// TIA Portal project "Trạm 4" (V17)

(* hardware
DEVICE "S7-1200 station_1"  S7-1200 Station
   slot 0: "Rack_0"  S7-1200 Rack  Rack  V1.0
   slot 1: "PLC_1"  CPU 1214C DC/DC/DC  6ES7 214-1AG40-0XB0  V4.4
*)

// ===== PLC "PLC_1"  CPU 1214C DC/DC/DC =====

VAR_GLOBAL   // PLC tag table "Default tag table"
   "Cảm biến phôi" AT %I0.0 : Bool;
   "Cảm biến vị trí gắp vật" AT %I0.1 : Bool;
   "Cảm biến vị trí trạm sau" AT %I0.2 : Bool;
   "Cảm biến vị trí khay" AT %I0.3 : Bool;
   "Cảm biến tay gắp xuống" AT %I0.4 : Bool;
   "Cảm biến tay gắp lên" AT %I0.5 : Bool;
   "CB_Mau" AT %I0.6 : Bool;
   "CB_TramIn" AT %I0.7 : Bool;
   "Start" AT %I1.0 : Bool;
   "Stop" AT %I1.1 : Bool;
   "Auto" AT %I1.2 : Bool;
   "Reset" AT %I1.3 : Bool;
   "HTTRai" AT %Q0.0 : Bool;
   "HTPhai" AT %Q0.1 : Bool;
   "Xi lanh xuống" AT %Q0.2 : Bool;
   "Kẹp phôi" AT %Q0.3 : Bool;
   "Yêu cầu cấp phôi" AT %Q0.7 : Bool;
   "LedStart" AT %Q1.0 : Bool;
   "LedReset" AT %Q1.1 : Bool;
   "TG_Start" AT %M0.0 : Bool;
   "TG_HTVat" AT %M0.1 : Bool;
   "TG_HTVat2" AT %M0.2 : Bool;
   "TG_TayGapXuong" AT %M0.3 : Bool;
   "TG_DungNhaVat" AT %M1.0 : Bool;
   "TG_CoVat" AT %M1.1 : Bool;
   "TG_Khay3" AT %M0.6 : Bool;
   "TG_HTkhay2" AT %M9.0 : Bool;
   "TG_CBHTV" AT %M9.1 : Bool;
   "TGCBVat" AT %M10.0 : Bool;
   "TG_ChoKep" AT %M0.4 : Bool;
   "TG_XilanhLen" AT %M0.5 : Bool;
   "TG_TramTiep" AT %M0.7 : Bool;
   "TG_XuongGapVat" AT %M1.2 : Bool;
   "TG_KepVat" AT %M1.3 : Bool;
   "TG_HTPhai" AT %M1.4 : Bool;
   "TG_DungTraVat" AT %M1.5 : Bool;
   "TG_NhaVat" AT %M1.6 : Bool;
   "TG_NhaVat2" AT %M1.7 : Bool;
   "TG_GapLoi" AT %M2.0 : Bool;
   "TG_Button_Reset" AT %M3.0 : Bool;
   "Tag_1" AT %M3.1 : Bool;
   "Tag_2" AT %M3.2 : Bool;
   "Tag_3" AT %M3.3 : Bool;
   "Tag_4" AT %M3.4 : Bool;
   "Tag_5" AT %M5.0 : Bool;
   "Tag_6" AT %M5.1 : Bool;
   "TG_Start_Manual" AT %M2.1 : Bool;
   "TG_Start_Auto" AT %M2.2 : Bool;
   "TG_TruyenThong_Reset" AT %M2.3 : Bool;
   "Reset_Truyen" AT %M2.4 : Bool;
END_VAR

VAR_GLOBAL   // PLC tag table "Trung gian tin hieu truyen nhan"
   "TG_PhoiThap" AT %M4.0 : Bool;
   "TG_PhoiCao" AT %M4.1 : Bool;
END_VAR

DATA_BLOCK "Data_TruyenThong05"   // DB31
{ S7_Optimized_Access := 'FALSE' }
VERSION : 0.1
   VAR
      Nhan_1 : Bool;
      Nhan_2 : Bool;
      Nhan_3 : Bool;
      Nhan_4 : Bool;
      Nhan_5 : Bool;
      Nhan_6 : Bool;
      Nhan_7 : Bool;
      Nhan_8 : Bool;
      truyen_1 : Bool;
      truyen_2 : Bool;
      truyen_3 : Bool;
      truyen_4 : Bool;
      truyen_5 : Bool;
      truyen_6 : Bool;
      truyen_7 : Bool;
      truyen_8 : Bool;
      truyen_9 : Bool;
      truyen_10 : Bool;
      truyen_11 : Bool;
      truyen_12 : Bool;
      truyen_13 : Bool;
      truyen_14 : Bool;
      truyen_15 : Bool;
      truyen_16 : Bool;
   END_VAR
BEGIN
END_DATA_BLOCK

// folder: System blocks/Program resources

DATA_BLOCK "Cho_Kep"   // DB26
{ S7_Optimized_Access := 'TRUE' }
AUTHOR : Simatic
FAMILY : IEC
NAME : IEC_TMR
VERSION : 1.0
// stored: InstanceOfName IEC_TIMER
"IEC_TIMER"
BEGIN
END_DATA_BLOCK

DATA_BLOCK "DungTraVat"   // DB27
{ S7_Optimized_Access := 'TRUE' }
AUTHOR : Simatic
FAMILY : IEC
NAME : IEC_TMR
VERSION : 1.0
// stored: InstanceOfName IEC_TIMER
"IEC_TIMER"
BEGIN
END_DATA_BLOCK

DATA_BLOCK "IEC_Timer_0_DB"   // DB28
{ S7_Optimized_Access := 'TRUE' }
AUTHOR : Simatic
FAMILY : IEC
NAME : IEC_TMR
VERSION : 1.0
// stored: InstanceOfName IEC_TIMER
"IEC_TIMER"
BEGIN
END_DATA_BLOCK

DATA_BLOCK "NhaVat_1"   // DB29
{ S7_Optimized_Access := 'TRUE' }
AUTHOR : Simatic
FAMILY : IEC
NAME : IEC_TMR
VERSION : 1.0
// stored: InstanceOfName IEC_TIMER
"IEC_TIMER"
BEGIN
END_DATA_BLOCK

DATA_BLOCK "TIme_GapVat"   // DB30
{ S7_Optimized_Access := 'TRUE' }
AUTHOR : Simatic
FAMILY : IEC
NAME : IEC_TMR
VERSION : 1.0
// stored: InstanceOfName IEC_TIMER
"IEC_TIMER"
BEGIN
END_DATA_BLOCK

// folder: (top level)

FUNCTION "GapVat" : Void   // FC1, LAD
{ S7_Optimized_Access := 'TRUE' }
VERSION : 0.1
BEGIN

REGION Network 1: Xác định có phôi ( Done ) -> CB phát hiện phôi + tay gắp ở vị trí trên + tay kẹp chưa kẹp = TG có phôi.
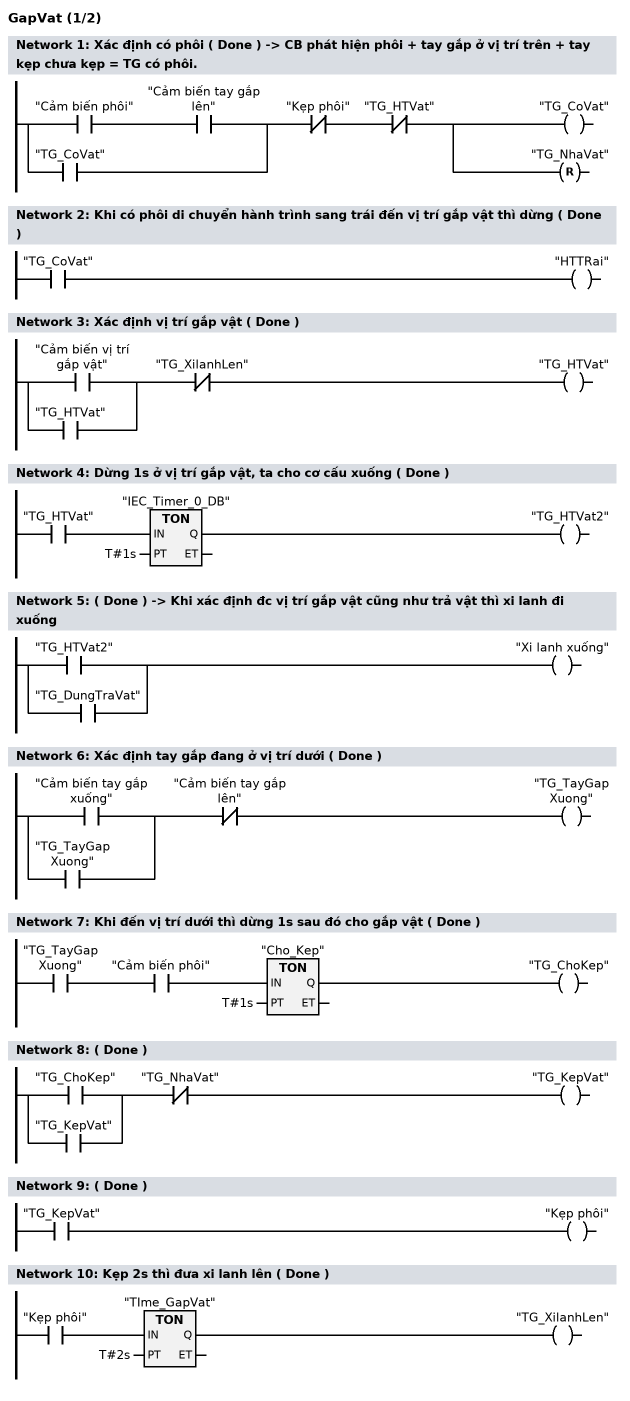
   RUNG wire#powerrail
      Contact( "Cảm biến phôi" )
      Contact( "Cảm biến tay gắp lên" )
      wire#w1
      I_Contact( "Kẹp phôi" )
      I_Contact( "TG_HTVat" )
      wire#w2
      Coil( "TG_CoVat" )
   END_RUNG
   RUNG wire#powerrail
      Contact( "TG_CoVat" )
   END_RUNG wire#w1
   RUNG wire#w2
      R_Coil( "TG_NhaVat" )
   END_RUNG
   // the same network as SCL:
   "TG_CoVat" := (("Cảm biến phôi" AND "Cảm biến tay gắp lên") OR "TG_CoVat") AND NOT "Kẹp phôi" AND NOT "TG_HTVat";
   IF "TG_CoVat" THEN "TG_NhaVat" := FALSE; END_IF;
END_REGION

REGION Network 2: Khi có phôi di chuyển hành trình sang trái đến vị trí gắp vật thì dừng ( Done )
   RUNG wire#powerrail
      Contact( "TG_CoVat" )
      Coil( "HTTRai" )
   END_RUNG
   // the same network as SCL:
   "HTTRai" := "TG_CoVat";
END_REGION

REGION Network 3: Xác định vị trí gắp vật ( Done )
   RUNG wire#powerrail
      Contact( "Cảm biến vị trí gắp vật" )
      wire#w1
      I_Contact( "TG_XilanhLen" )
      Coil( "TG_HTVat" )
   END_RUNG
   RUNG wire#powerrail
      Contact( "TG_HTVat" )
   END_RUNG wire#w1
   // the same network as SCL:
   "TG_HTVat" := ("Cảm biến vị trí gắp vật" OR "TG_HTVat") AND NOT "TG_XilanhLen";
END_REGION

REGION Network 4: Dừng 1s ở vị trí gắp vật, ta cho cơ cấu xuống ( Done )
   "IEC_Timer_0_DB".TON(IN := "TG_HTVat", PT := T#1s);
   "TG_HTVat2" := "IEC_Timer_0_DB".Q;
END_REGION

REGION Network 5: ( Done ) -> Khi xác định đc vị trí gắp vật cũng như trả vật thì xi lanh đi xuống
   RUNG wire#powerrail
      Contact( "TG_HTVat2" )
      wire#w1
      Coil( "Xi lanh xuống" )
   END_RUNG
   RUNG wire#powerrail
      Contact( "TG_DungTraVat" )
   END_RUNG wire#w1
   // the same network as SCL:
   "Xi lanh xuống" := "TG_HTVat2" OR "TG_DungTraVat";
END_REGION

REGION Network 6: Xác định tay gắp đang ở vị trí dưới ( Done )
   RUNG wire#powerrail
      Contact( "Cảm biến tay gắp xuống" )
      wire#w1
      I_Contact( "Cảm biến tay gắp lên" )
      Coil( "TG_TayGapXuong" )
   END_RUNG
   RUNG wire#powerrail
      Contact( "TG_TayGapXuong" )
   END_RUNG wire#w1
   // the same network as SCL:
   "TG_TayGapXuong" := ("Cảm biến tay gắp xuống" OR "TG_TayGapXuong") AND NOT "Cảm biến tay gắp lên";
END_REGION

REGION Network 7: Khi đến vị trí dưới thì dừng 1s sau đó cho gắp vật ( Done )
   "Cho_Kep".TON(IN := "TG_TayGapXuong" AND "Cảm biến phôi", PT := T#1s);
   "TG_ChoKep" := "Cho_Kep".Q;
END_REGION

REGION Network 8: ( Done )
   RUNG wire#powerrail
      Contact( "TG_ChoKep" )
      wire#w1
      I_Contact( "TG_NhaVat" )
      Coil( "TG_KepVat" )
   END_RUNG
   RUNG wire#powerrail
      Contact( "TG_KepVat" )
   END_RUNG wire#w1
   // the same network as SCL:
   "TG_KepVat" := ("TG_ChoKep" OR "TG_KepVat") AND NOT "TG_NhaVat";
END_REGION

REGION Network 9: ( Done )
   RUNG wire#powerrail
      Contact( "TG_KepVat" )
      Coil( "Kẹp phôi" )
   END_RUNG
   // the same network as SCL:
   "Kẹp phôi" := "TG_KepVat";
END_REGION

REGION Network 10: Kẹp 2s thì đưa xi lanh lên ( Done )
   "TIme_GapVat".TON(IN := "Kẹp phôi", PT := T#2s);
   "TG_XilanhLen" := "TIme_GapVat".Q;
END_REGION

REGION Network 11: Khi xi lanh ở vị tri trên và đang kẹp vật thì cho sang phải ( Done )
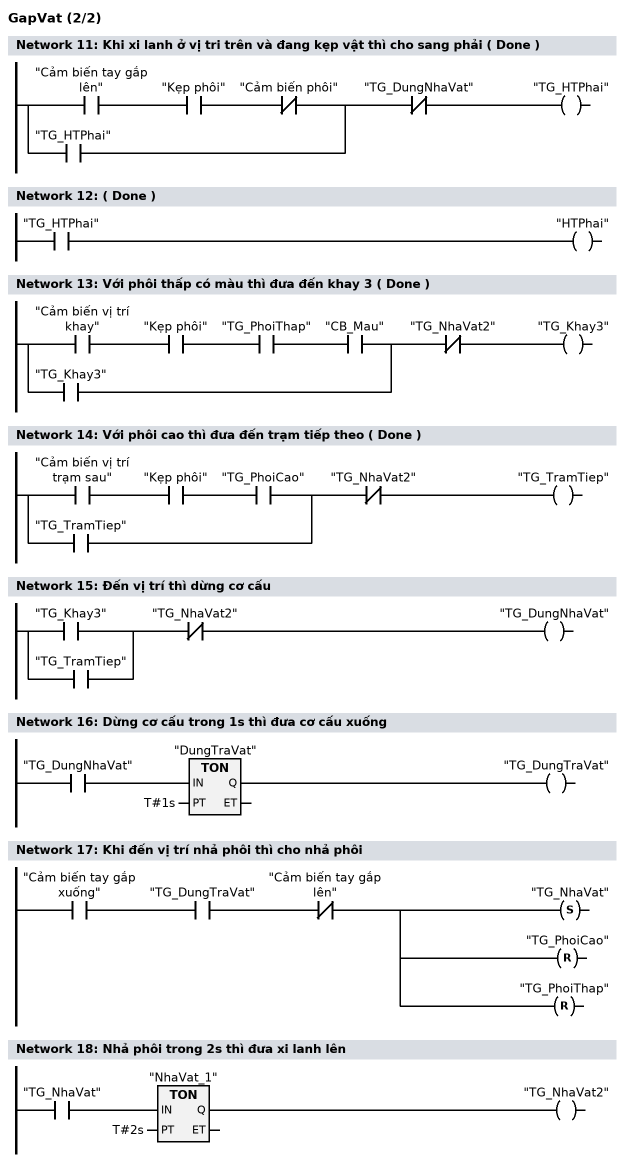
   RUNG wire#powerrail
      Contact( "Cảm biến tay gắp lên" )
      Contact( "Kẹp phôi" )
      I_Contact( "Cảm biến phôi" )
      wire#w1
      I_Contact( "TG_DungNhaVat" )
      Coil( "TG_HTPhai" )
   END_RUNG
   RUNG wire#powerrail
      Contact( "TG_HTPhai" )
   END_RUNG wire#w1
   // the same network as SCL:
   "TG_HTPhai" := (("Cảm biến tay gắp lên" AND "Kẹp phôi" AND NOT "Cảm biến phôi") OR "TG_HTPhai") AND NOT "TG_DungNhaVat";
END_REGION

REGION Network 12: ( Done )
   RUNG wire#powerrail
      Contact( "TG_HTPhai" )
      Coil( "HTPhai" )
   END_RUNG
   // the same network as SCL:
   "HTPhai" := "TG_HTPhai";
END_REGION

REGION Network 13: Với phôi thấp có màu thì đưa đến khay 3 ( Done )
   RUNG wire#powerrail
      Contact( "Cảm biến vị trí khay" )
      Contact( "Kẹp phôi" )
      Contact( "TG_PhoiThap" )
      Contact( "CB_Mau" )
      wire#w1
      I_Contact( "TG_NhaVat2" )
      Coil( "TG_Khay3" )
   END_RUNG
   RUNG wire#powerrail
      Contact( "TG_Khay3" )
   END_RUNG wire#w1
   // the same network as SCL:
   "TG_Khay3" := (("Cảm biến vị trí khay" AND "Kẹp phôi" AND "TG_PhoiThap" AND "CB_Mau") OR "TG_Khay3") AND NOT "TG_NhaVat2";
END_REGION

REGION Network 14: Với phôi cao thì đưa đến trạm tiếp theo ( Done )
   RUNG wire#powerrail
      Contact( "Cảm biến vị trí trạm sau" )
      Contact( "Kẹp phôi" )
      Contact( "TG_PhoiCao" )
      wire#w1
      I_Contact( "TG_NhaVat2" )
      Coil( "TG_TramTiep" )
   END_RUNG
   RUNG wire#powerrail
      Contact( "TG_TramTiep" )
   END_RUNG wire#w1
   // the same network as SCL:
   "TG_TramTiep" := (("Cảm biến vị trí trạm sau" AND "Kẹp phôi" AND "TG_PhoiCao") OR "TG_TramTiep") AND NOT "TG_NhaVat2";
END_REGION

REGION Network 15: Đến vị trí thì dừng cơ cấu
   RUNG wire#powerrail
      Contact( "TG_Khay3" )
      wire#w1
      I_Contact( "TG_NhaVat2" )
      Coil( "TG_DungNhaVat" )
   END_RUNG
   RUNG wire#powerrail
      Contact( "TG_TramTiep" )
   END_RUNG wire#w1
   // the same network as SCL:
   "TG_DungNhaVat" := ("TG_Khay3" OR "TG_TramTiep") AND NOT "TG_NhaVat2";
END_REGION

REGION Network 16: Dừng cơ cấu trong 1s thì đưa cơ cấu xuống
   "DungTraVat".TON(IN := "TG_DungNhaVat", PT := T#1s);
   "TG_DungTraVat" := "DungTraVat".Q;
END_REGION

REGION Network 17: Khi đến vị trí nhả phôi thì cho nhả phôi
   RUNG wire#powerrail
      Contact( "Cảm biến tay gắp xuống" )
      Contact( "TG_DungTraVat" )
      I_Contact( "Cảm biến tay gắp lên" )
      wire#w1
      S_Coil( "TG_NhaVat" )
   END_RUNG
   RUNG wire#w1
      R_Coil( "TG_PhoiCao" )
   END_RUNG
   RUNG wire#w1
      R_Coil( "TG_PhoiThap" )
   END_RUNG
   // the same network as SCL:
   IF "Cảm biến tay gắp xuống" AND "TG_DungTraVat" AND NOT "Cảm biến tay gắp lên" THEN
       "TG_NhaVat" := TRUE;
       "TG_PhoiCao" := FALSE;
       "TG_PhoiThap" := FALSE;
   END_IF;
END_REGION

REGION Network 18: Nhả phôi trong 2s thì đưa xi lanh lên
   "NhaVat_1".TON(IN := "TG_NhaVat", PT := T#2s);
   "TG_NhaVat2" := "NhaVat_1".Q;
END_REGION
END_FUNCTION

FUNCTION "OBReset" : Void   // FC2, LAD
{ S7_Optimized_Access := 'TRUE' }
VERSION : 0.1
   VAR_TEMP   // added for the SCL form of the ladder/FBD networks
      _w1 : Bool;
   END_VAR
BEGIN

REGION Network 1: Reset các trạng thái
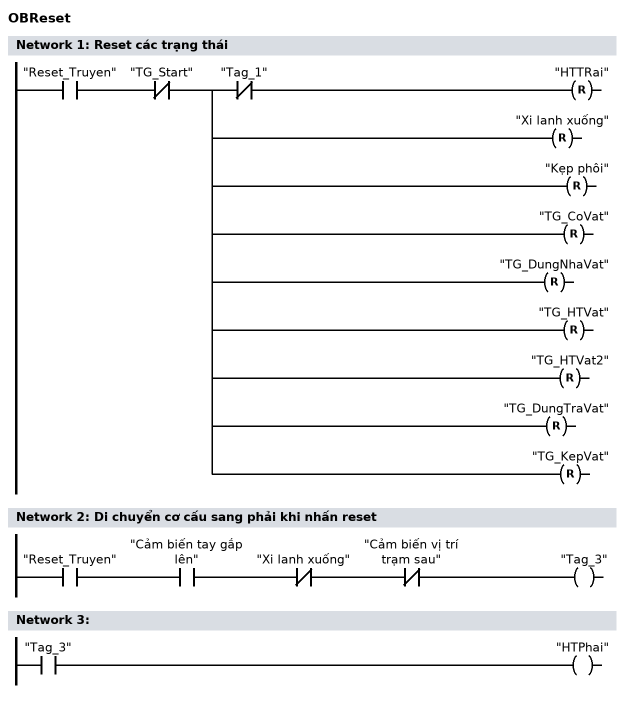
   RUNG wire#powerrail
      Contact( "Reset_Truyen" )
      I_Contact( "TG_Start" )
      wire#w1
      I_Contact( "Tag_1" )
      R_Coil( "HTTRai" )
   END_RUNG
   RUNG wire#w1
      R_Coil( "Xi lanh xuống" )
   END_RUNG
   RUNG wire#w1
      R_Coil( "Kẹp phôi" )
   END_RUNG
   RUNG wire#w1
      R_Coil( "TG_CoVat" )
   END_RUNG
   RUNG wire#w1
      R_Coil( "TG_DungNhaVat" )
   END_RUNG
   RUNG wire#w1
      R_Coil( "TG_HTVat" )
   END_RUNG
   RUNG wire#w1
      R_Coil( "TG_HTVat2" )
   END_RUNG
   RUNG wire#w1
      R_Coil( "TG_DungTraVat" )
   END_RUNG
   RUNG wire#w1
      R_Coil( "TG_KepVat" )
   END_RUNG
   // the same network as SCL:
   #_w1 := "Reset_Truyen" AND NOT "TG_Start";
   IF #_w1 AND NOT "Tag_1" THEN "HTTRai" := FALSE; END_IF;
   IF #_w1 THEN
       "Xi lanh xuống" := FALSE;
       "Kẹp phôi" := FALSE;
       "TG_CoVat" := FALSE;
       "TG_DungNhaVat" := FALSE;
       "TG_HTVat" := FALSE;
       "TG_HTVat2" := FALSE;
       "TG_DungTraVat" := FALSE;
       "TG_KepVat" := FALSE;
   END_IF;
END_REGION

REGION Network 2: Di chuyển cơ cấu sang phải khi nhấn reset
   RUNG wire#powerrail
      Contact( "Reset_Truyen" )
      Contact( "Cảm biến tay gắp lên" )
      I_Contact( "Xi lanh xuống" )
      I_Contact( "Cảm biến vị trí trạm sau" )
      Coil( "Tag_3" )
   END_RUNG
   // the same network as SCL:
   "Tag_3" := "Reset_Truyen" AND "Cảm biến tay gắp lên" AND NOT "Xi lanh xuống" AND NOT "Cảm biến vị trí trạm sau";
END_REGION

REGION Network 3
   RUNG wire#powerrail
      Contact( "Tag_3" )
      Coil( "HTPhai" )
   END_RUNG
   // the same network as SCL:
   "HTPhai" := "Tag_3";
END_REGION
END_FUNCTION

ORGANIZATION_BLOCK "Main"   // OB1, LAD, ProgramCycle
TITLE = "Main Program Sweep (Cycle)"
{ S7_Optimized_Access := 'TRUE' }
VERSION : 0.1
   VAR_INPUT
      Initial_Call : Bool;   // Initial call of this OB
      Remanence : Bool;   // =True, if remanent data are available
   END_VAR
BEGIN

REGION Network 1: Trạng thái Start ở chế độ Manual ( Done ) -> Vặn khóa + ấn Start và k có tín hiệu Auto từ HMI = Manual
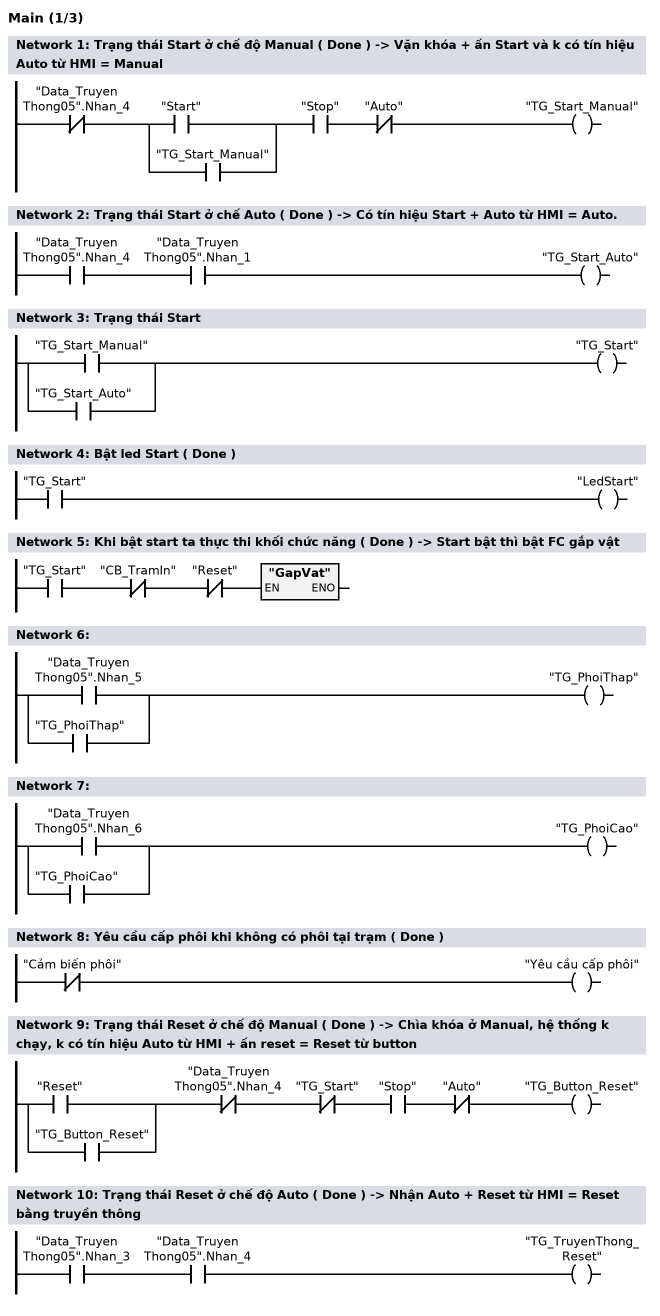
   RUNG wire#powerrail
      I_Contact( "Data_TruyenThong05".Nhan_4 )
      wire#w1
      Contact( "Start" )
      wire#w2
      Contact( "Stop" )
      I_Contact( "Auto" )
      Coil( "TG_Start_Manual" )
   END_RUNG
   RUNG wire#w1
      Contact( "TG_Start_Manual" )
   END_RUNG wire#w2
   // the same network as SCL:
   "TG_Start_Manual" := NOT "Data_TruyenThong05".Nhan_4 AND ("Start" OR "TG_Start_Manual") AND "Stop" AND NOT "Auto";
END_REGION

REGION Network 2: Trạng thái Start ở chế Auto ( Done ) -> Có tín hiệu Start + Auto từ HMI = Auto.
   RUNG wire#powerrail
      Contact( "Data_TruyenThong05".Nhan_4 )
      Contact( "Data_TruyenThong05".Nhan_1 )
      Coil( "TG_Start_Auto" )
   END_RUNG
   // the same network as SCL:
   "TG_Start_Auto" := "Data_TruyenThong05".Nhan_4 AND "Data_TruyenThong05".Nhan_1;
END_REGION

REGION Network 3: Trạng thái Start
   RUNG wire#powerrail
      Contact( "TG_Start_Manual" )
      wire#w1
      Coil( "TG_Start" )
   END_RUNG
   RUNG wire#powerrail
      Contact( "TG_Start_Auto" )
   END_RUNG wire#w1
   // the same network as SCL:
   "TG_Start" := "TG_Start_Manual" OR "TG_Start_Auto";
END_REGION

REGION Network 4: Bật led Start ( Done )
   RUNG wire#powerrail
      Contact( "TG_Start" )
      Coil( "LedStart" )
   END_RUNG
   // the same network as SCL:
   "LedStart" := "TG_Start";
END_REGION

REGION Network 5: Khi bật start ta thực thi khối chức năng ( Done ) -> Start bật thì bật FC gắp vật
   RUNG wire#powerrail
      Contact( "TG_Start" )
      I_Contact( "CB_TramIn" )
      I_Contact( "Reset" )
      "GapVat"()
   END_RUNG
   // the same network as SCL:
   IF "TG_Start" AND NOT "CB_TramIn" AND NOT "Reset" THEN "GapVat"(); END_IF;
END_REGION

REGION Network 6
   RUNG wire#powerrail
      Contact( "Data_TruyenThong05".Nhan_5 )
      wire#w1
      Coil( "TG_PhoiThap" )
   END_RUNG
   RUNG wire#powerrail
      Contact( "TG_PhoiThap" )
   END_RUNG wire#w1
   // the same network as SCL:
   "TG_PhoiThap" := "Data_TruyenThong05".Nhan_5 OR "TG_PhoiThap";
END_REGION

REGION Network 7
   RUNG wire#powerrail
      Contact( "Data_TruyenThong05".Nhan_6 )
      wire#w1
      Coil( "TG_PhoiCao" )
   END_RUNG
   RUNG wire#powerrail
      Contact( "TG_PhoiCao" )
   END_RUNG wire#w1
   // the same network as SCL:
   "TG_PhoiCao" := "Data_TruyenThong05".Nhan_6 OR "TG_PhoiCao";
END_REGION

REGION Network 8: Yêu cầu cấp phôi khi không có phôi tại trạm ( Done )
   RUNG wire#powerrail
      I_Contact( "Cảm biến phôi" )
      Coil( "Yêu cầu cấp phôi" )
   END_RUNG
   // the same network as SCL:
   "Yêu cầu cấp phôi" := NOT "Cảm biến phôi";
END_REGION

REGION Network 9: Trạng thái Reset ở chế độ Manual ( Done ) -> Chìa khóa ở Manual, hệ thống k chạy, k có tín hiệu Auto từ HMI + ấn reset = Reset từ button
   RUNG wire#powerrail
      Contact( "Reset" )
      wire#w1
      I_Contact( "Data_TruyenThong05".Nhan_4 )
      I_Contact( "TG_Start" )
      Contact( "Stop" )
      I_Contact( "Auto" )
      Coil( "TG_Button_Reset" )
   END_RUNG
   RUNG wire#powerrail
      Contact( "TG_Button_Reset" )
   END_RUNG wire#w1
   // the same network as SCL:
   "TG_Button_Reset" := ("Reset" OR "TG_Button_Reset") AND NOT "Data_TruyenThong05".Nhan_4 AND NOT "TG_Start" AND "Stop" AND NOT "Auto";
END_REGION

REGION Network 10: Trạng thái Reset ở chế độ Auto ( Done ) -> Nhận Auto + Reset từ HMI = Reset bằng truyền thông
   RUNG wire#powerrail
      Contact( "Data_TruyenThong05".Nhan_3 )
      Contact( "Data_TruyenThong05".Nhan_4 )
      Coil( "TG_TruyenThong_Reset" )
   END_RUNG
   // the same network as SCL:
   "TG_TruyenThong_Reset" := "Data_TruyenThong05".Nhan_3 AND "Data_TruyenThong05".Nhan_4;
END_REGION

REGION Network 11: Trạng thái Reset ( Done )
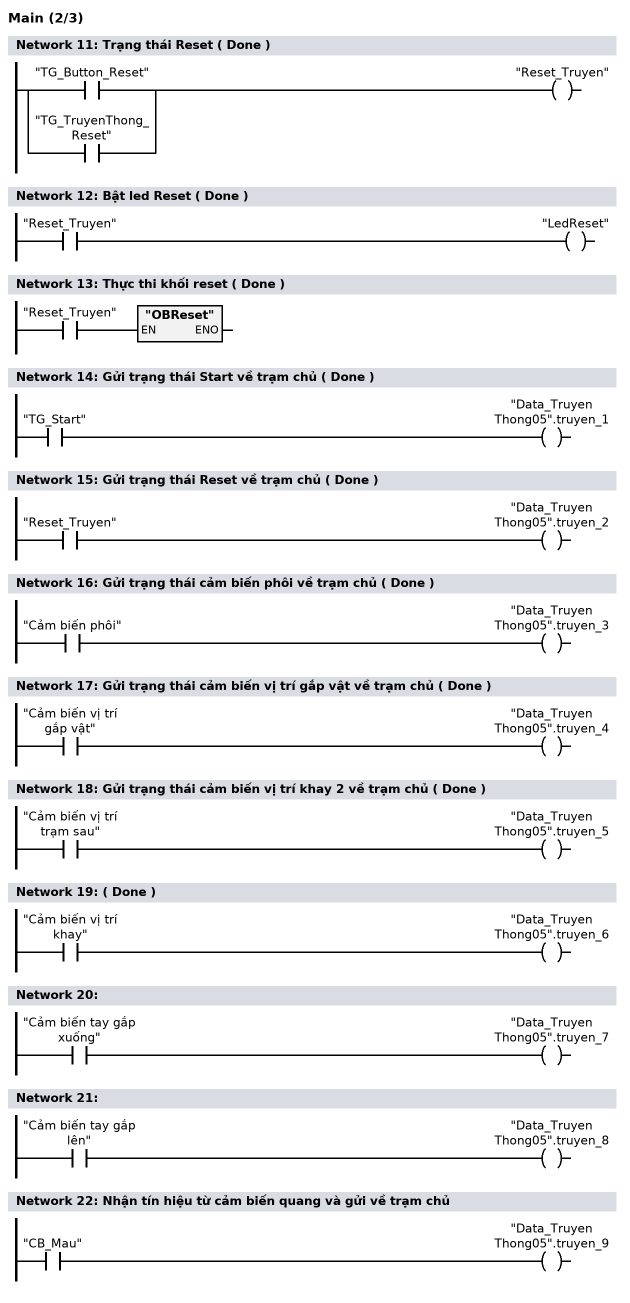
   RUNG wire#powerrail
      Contact( "TG_Button_Reset" )
      wire#w1
      Coil( "Reset_Truyen" )
   END_RUNG
   RUNG wire#powerrail
      Contact( "TG_TruyenThong_Reset" )
   END_RUNG wire#w1
   // the same network as SCL:
   "Reset_Truyen" := "TG_Button_Reset" OR "TG_TruyenThong_Reset";
END_REGION

REGION Network 12: Bật led Reset ( Done )
   RUNG wire#powerrail
      Contact( "Reset_Truyen" )
      Coil( "LedReset" )
   END_RUNG
   // the same network as SCL:
   "LedReset" := "Reset_Truyen";
END_REGION

REGION Network 13: Thực thi khối reset ( Done )
   RUNG wire#powerrail
      Contact( "Reset_Truyen" )
      "OBReset"()
   END_RUNG
   // the same network as SCL:
   IF "Reset_Truyen" THEN "OBReset"(); END_IF;
END_REGION

REGION Network 14: Gửi trạng thái Start về trạm chủ ( Done )
   RUNG wire#powerrail
      Contact( "TG_Start" )
      Coil( "Data_TruyenThong05".truyen_1 )
   END_RUNG
   // the same network as SCL:
   "Data_TruyenThong05".truyen_1 := "TG_Start";
END_REGION

REGION Network 15: Gửi trạng thái Reset về trạm chủ ( Done )
   RUNG wire#powerrail
      Contact( "Reset_Truyen" )
      Coil( "Data_TruyenThong05".truyen_2 )
   END_RUNG
   // the same network as SCL:
   "Data_TruyenThong05".truyen_2 := "Reset_Truyen";
END_REGION

REGION Network 16: Gửi trạng thái cảm biến phôi về trạm chủ ( Done )
   RUNG wire#powerrail
      Contact( "Cảm biến phôi" )
      Coil( "Data_TruyenThong05".truyen_3 )
   END_RUNG
   // the same network as SCL:
   "Data_TruyenThong05".truyen_3 := "Cảm biến phôi";
END_REGION

REGION Network 17: Gửi trạng thái cảm biến vị trí gắp vật về trạm chủ ( Done )
   RUNG wire#powerrail
      Contact( "Cảm biến vị trí gắp vật" )
      Coil( "Data_TruyenThong05".truyen_4 )
   END_RUNG
   // the same network as SCL:
   "Data_TruyenThong05".truyen_4 := "Cảm biến vị trí gắp vật";
END_REGION

REGION Network 18: Gửi trạng thái cảm biến vị trí khay 2 về trạm chủ ( Done )
   RUNG wire#powerrail
      Contact( "Cảm biến vị trí trạm sau" )
      Coil( "Data_TruyenThong05".truyen_5 )
   END_RUNG
   // the same network as SCL:
   "Data_TruyenThong05".truyen_5 := "Cảm biến vị trí trạm sau";
END_REGION

REGION Network 19: ( Done )
   RUNG wire#powerrail
      Contact( "Cảm biến vị trí khay" )
      Coil( "Data_TruyenThong05".truyen_6 )
   END_RUNG
   // the same network as SCL:
   "Data_TruyenThong05".truyen_6 := "Cảm biến vị trí khay";
END_REGION

REGION Network 20
   RUNG wire#powerrail
      Contact( "Cảm biến tay gắp xuống" )
      Coil( "Data_TruyenThong05".truyen_7 )
   END_RUNG
   // the same network as SCL:
   "Data_TruyenThong05".truyen_7 := "Cảm biến tay gắp xuống";
END_REGION

REGION Network 21
   RUNG wire#powerrail
      Contact( "Cảm biến tay gắp lên" )
      Coil( "Data_TruyenThong05".truyen_8 )
   END_RUNG
   // the same network as SCL:
   "Data_TruyenThong05".truyen_8 := "Cảm biến tay gắp lên";
END_REGION

REGION Network 22: Nhận tín hiệu từ cảm biến quang và gửi về trạm chủ
   RUNG wire#powerrail
      Contact( "CB_Mau" )
      Coil( "Data_TruyenThong05".truyen_9 )
   END_RUNG
   // the same network as SCL:
   "Data_TruyenThong05".truyen_9 := "CB_Mau";
END_REGION

REGION Network 23: Nhận tín hiệu từ trạm sau và gửi trạm chủ
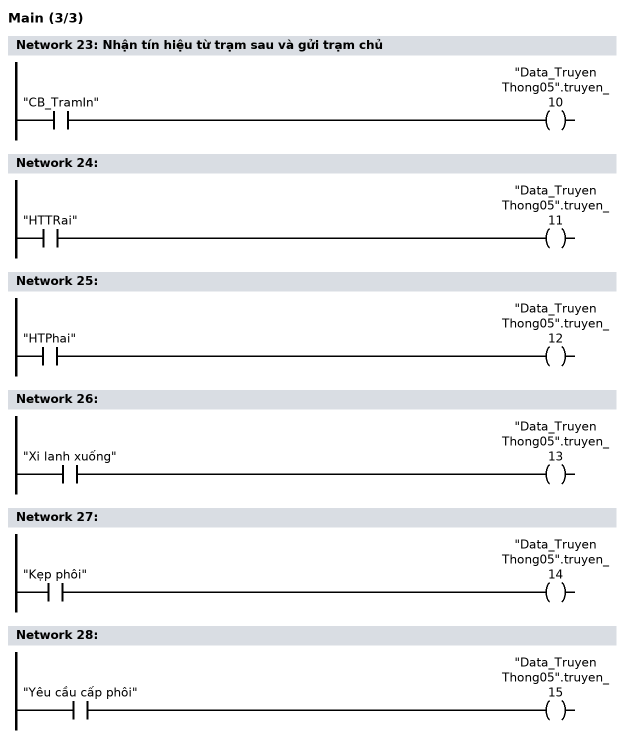
   RUNG wire#powerrail
      Contact( "CB_TramIn" )
      Coil( "Data_TruyenThong05".truyen_10 )
   END_RUNG
   // the same network as SCL:
   "Data_TruyenThong05".truyen_10 := "CB_TramIn";
END_REGION

REGION Network 24
   RUNG wire#powerrail
      Contact( "HTTRai" )
      Coil( "Data_TruyenThong05".truyen_11 )
   END_RUNG
   // the same network as SCL:
   "Data_TruyenThong05".truyen_11 := "HTTRai";
END_REGION

REGION Network 25
   RUNG wire#powerrail
      Contact( "HTPhai" )
      Coil( "Data_TruyenThong05".truyen_12 )
   END_RUNG
   // the same network as SCL:
   "Data_TruyenThong05".truyen_12 := "HTPhai";
END_REGION

REGION Network 26
   RUNG wire#powerrail
      Contact( "Xi lanh xuống" )
      Coil( "Data_TruyenThong05".truyen_13 )
   END_RUNG
   // the same network as SCL:
   "Data_TruyenThong05".truyen_13 := "Xi lanh xuống";
END_REGION

REGION Network 27
   RUNG wire#powerrail
      Contact( "Kẹp phôi" )
      Coil( "Data_TruyenThong05".truyen_14 )
   END_RUNG
   // the same network as SCL:
   "Data_TruyenThong05".truyen_14 := "Kẹp phôi";
END_REGION

REGION Network 28
   RUNG wire#powerrail
      Contact( "Yêu cầu cấp phôi" )
      Coil( "Data_TruyenThong05".truyen_15 )
   END_RUNG
   // the same network as SCL:
   "Data_TruyenThong05".truyen_15 := "Yêu cầu cấp phôi";
END_REGION
END_ORGANIZATION_BLOCK